{attribute 'GeneratedUsingTerminal: EK1100-0000-0018'}
{attribute addProperty BoxType "EK1100-0000-0018"}
{attribute addProperty Id "Beckhoff_AT2xxxEK1122Beckhoff_AT2xxxEK1122_43DD63D75810A_0059_AT2000_5250_0018AT2000_33A3DF1B80"}
{attribute addProperty CRC "666313065"}
{attribute addProperty Size "5890"}
{attribute addProperty Name "Beckhoff AT1xxx"}
TYPE Beckhoff_AT1xxx_27B72169 EXTENDS EK1100_1FC0878B :
STRUCT
	{attribute addProperty Name "Beckhoff AT2xxxEK1122"}
	{attribute addProperty PreviousPort "Beckhoff AT1xxx : B"}
	Beckhoff_AT2xxxEK1122 : Beckhoff_AT2xxxEK1122_43DD63D7;
	{attribute addProperty Name "A_0059(AT2000-5250-0018)"}
	{attribute addProperty PreviousPort "Beckhoff AT2xxxEK1122 : C"}
	A_0059_AT2000_5250_0018 : AT2000_33A3DF1B;
END_STRUCT
END_TYPE

(* stored: Version 1.2.0.0, ProductVersion 3.1.4024.11
   DUT Beckhoff_AT1xxx_27B72169: Id {f6e879c4-f7eb-49c2-98ea-17ddb61d1fd9} *)
